// LS Electric XG5000 project: test
// PLC NewPLC

PROGRAM NewProgram (task: 스캔 프로그램)

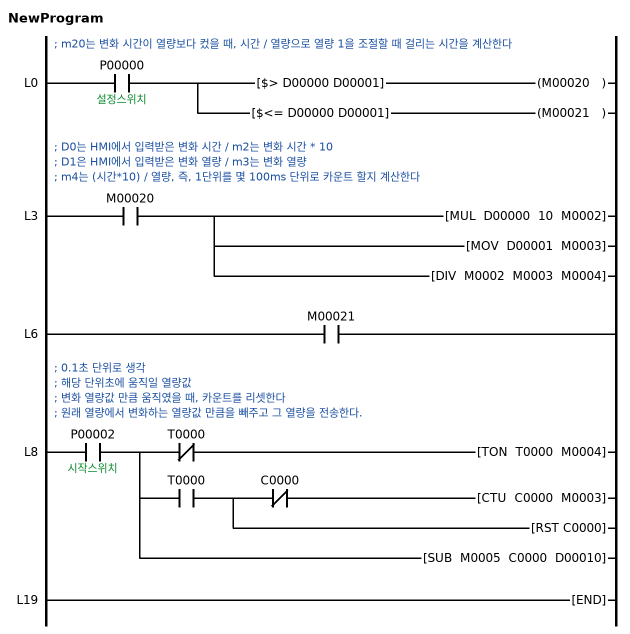
; L0
// network not rendered as a mnemonic list; see the picture
// output comment: m20는 변화 시간이 열량보다 컸을 때, 시간 / 열량으로 열량 1을 조절할 때 걸리는 시간을 계산한다
; L3
LOAD      M00020
MUL       D00000 10 M0002
MOV       D00001 M0003
DIV       M0002 M0003 M0004
// output comment: D0는 HMI에서 입력받은 변화 시간 / m2는 변화 시간 * 10
// output comment: D1은 HMI에서 입력받은 변화 열량 / m3는 변화 열량
// output comment: m4는 (시간*10) / 열량, 즉, 1단위를 몇 100ms 단위로 카운트 할지 계산한다
; L6
LOAD      M00021
; L8
LOAD      P00002	// 시작스위치
MPUSH
AND NOT   T0000
TON       T0000 M0004
MLOAD
AND       T0000
MPUSH
AND NOT   C0000
CTU       C0000 M0003
MPOP
RST       C0000
MPOP
SUB       M0005 C0000 D00010
// output comment: 0.1초 단위로 생각
// output comment: 해당 단위초에 움직일 열량값
// output comment: 변화 열량값 만큼 움직였을 때, 카운트를 리셋한다
// output comment: 원래 열량에서 변화하는 열량값 만큼을 빼주고 그 열량을 전송한다.
; L19
END